{attribute 'GeneratedUsingTerminal: ELX3202-0000-0016'}
{attribute addProperty BoxType "ELX3202-0000-0016"}
{attribute addProperty Id "StatusAT %I*Status_F2CE6D917ValueAT %I*INT2"}
{attribute addProperty CRC "1245267073"}
{attribute addProperty Size "9"}
TYPE RTD_Inputs_Channel_4A394481 :
STRUCT
	{attribute addProperty Name "Status"}
	Status AT %I* : Status_F2CE6D91;
	{attribute addProperty Name "Value"}
	Value AT %I* : INT;
END_STRUCT
END_TYPE

(* stored: Version 1.2.0.0, ProductVersion 3.1.4024.9
   DUT RTD_Inputs_Channel_4A394481: Id {f39b7c05-20d6-4c97-b666-f11f9a7d2ade} *)
